{attribute 'linkalways'} 
{attribute 'no_explicit_call' := 'This FB is a CLASS and must be accessed using methods or properties'}
{attribute 'enable_dynamic_creation'}
FUNCTION_BLOCK Node_F_VN_FillContainer_UDINT EXTENDS VisionNode
VAR
    ipContainer : _ITcVnContainer;
    nValue : _UDINT(0);
    hrPrev : _HRESULT(S_OK);
    hresult : _HRESULT(S_OK);
END_VAR

METHOD PUBLIC  Clone : I_Node
VAR
    pNode : POINTER TO Node_F_VN_FillContainer_UDINT;
END_VAR
pNode := __NEW(Node_F_VN_FillContainer_UDINT);
Clone := pNode^;
END_METHOD

METHOD FB_init : BOOL
VAR_INPUT
    bInitRetains : BOOL; // if TRUE, the retain variables are initialized (warm start / cold start)
    bInCopyCode : BOOL;  // if TRUE, the instance afterwards gets moved into the copy code (online change)
END_VAR
AddInput('ipContainer', ipContainer);
AddInput('nValue', nValue);
AddInput('hrPrev', hrPrev);
AddOutput('ipContainer', ipContainer);
AddOutput('hresult',hresult);
END_METHOD

METHOD PROTECTED OnExecute : HRESULT
hresult.Value := F_VN_FillContainer_UDINT(
    ipContainer := ipContainer.Value,
    nValue := nValue.Value,
    hrPrev:= hrPrev.Value);
END_METHOD

METHOD PUBLIC PreExecutionCheck
VAR_INPUT
    Check : I_PreExecutionChecks;
END_VAR
Check.IsTrue(ipContainer.IsValid, 'ipContainer must be a valid container');
END_METHOD

END_FUNCTION_BLOCK

(* stored: Version 1.1.0.1, ProductVersion 3.1.4024.13
   POU Node_F_VN_FillContainer_UDINT: Id {9ac324d5-d6fb-4d43-bbf4-fea95854fec2}, SpecialFunc None
   Folder Constructor: Id {4f19bda4-9b65-43da-8ae6-8cc088eb6a0a}
   Method Clone: Id {ee844e21-2f11-49c1-855c-7028a9789df4}
   Method FB_init: Id {1ef8f110-ae59-44ac-8942-4fc23dc578d4}
   Method OnExecute: Id {ac2b81b0-94c0-4ddb-ba10-e98fce112693}
   Method PreExecutionCheck: Id {45f92643-b3d9-4dff-9491-0049c912cd97} *)
